FUNCTION_BLOCK PUBLIC FB_Observable IMPLEMENTS I_Observable
VAR_INPUT
	iParent:		I_Element;	
END_VAR
VAR
	bObserver:		BOOL;
	pList: 			POINTER TO I_Element;
    {attribute 'hide'}
	nLength:		DINT;
	{IF (defined (release))}
    	{attribute 'hide'}
	{END_IF}
	aList:			POINTER TO POINTER TO ARRAY [0..100] OF I_Element:=ADR(pList);
END_VAR

// https://peterzerlauth.com/
bObserver:= TRUE;

METHOD FB_exit : BOOL
VAR_INPUT
	bInCopyCode : BOOL; // if TRUE, the exit method is called for exiting an instance that is copied afterwards (online change).
END_VAR
M_Clear();
END_METHOD

METHOD M_Attach : BOOL
VAR_INPUT
	iObject: 	I_Element;
END_VAR
VAR
	pOldList: 	POINTER TO I_Element;
END_VAR
IF iObject <> 0 THEN
	// First Item
	IF pList = 0 THEN
		nLength:= nLength + 1;
		pList:= __NEW(POINTER TO I_Element,DINT_TO_UDINT(nLength));
	ELSE
		// Item already in List
		IF M_Find(iObject) = -1 THEN
			// backup 
			pOldList:= pList;
			// new Length
			nLength:= nLength + 1;
			// new pointer
			pList:= __NEW(POINTER TO I_Element,DINT_TO_UDINT(nLength));
			// restore
			Memcpy(pList,pOldList, SIZEOF(POINTER TO I_Element)*DINT_TO_UDINT(nLength -1));
			// delete old
			__DELETE(pOldList);
		ELSE
			M_Attach:= FALSE;	
			RETURN;
		END_IF
	END_IF
	IF pList = 0 THEN
		RETURN;
	END_IF
	// add new Object
	pList[nLength-1]:= iObject;
	M_Attach:= TRUE;
ELSE
	M_Attach:= FALSE;	
END_IF
END_METHOD

METHOD M_Clear
IF pList <> 0 THEN
	nLength:= 0;
	__DELETE(pList);
END_IF
END_METHOD

METHOD M_Detach : BOOL
VAR_INPUT
	iObject: 	I_Element;
END_VAR
VAR
	pOldList:			POINTER TO I_Element;
	nPosition: 			DINT;
END_VAR
IF iObject <> 0 THEN
	// First Item
	IF nLength >= 0 THEN
		// Item already in List
		nPosition:= M_Find(iObject);
		IF nPosition <> -1 THEN
			// backup 
			pOldList:= pList;
			// new Length
			nLength:= nLength -1;
			// new pointer
			pList:= __NEW(POINTER TO I_Element,DINT_TO_UDINT(nLength));
			// restore lower part
			Memcpy(pList,pOldList, SIZEOF(POINTER TO I_Element) * DINT_TO_UDINT(nPosition));
			//pList[nPosition]:= iObject;
			Memcpy(pList + (SIZEOF(POINTER TO I_Element)*nPosition),pOldList + (SIZEOF(POINTER TO I_Element)*(nPosition + 1)), SIZEOF(POINTER TO I_Element) * DINT_TO_UDINT(nLength - nPosition));
			// delete old
			__DELETE(pOldList);
		ELSE
			M_Detach:= FALSE;	
			RETURN;
		END_IF
	ELSE
		M_Detach:= FALSE;	
		RETURN;
	END_IF
	M_Detach:= TRUE;
ELSE
	M_Detach:= FALSE;	
END_IF
END_METHOD

METHOD M_Find : DINT
VAR_INPUT
	iObject: 	I_Element;
END_VAR
VAR
	nIndex: 	UINT;
END_VAR
// Object already in List
M_Find := -1;
WHILE nIndex < nLength DO
    IF (pList[nIndex] = iObject) THEN
        M_Find := nIndex;
        RETURN;
    END_IF
	nIndex := nIndex + 1;
END_WHILE
END_METHOD

METHOD M_Index : I_Observer
VAR_INPUT
	nIndex: 	DINT;
END_VAR
IF nIndex <= nLength THEN
	M_Index:= pList[nIndex].P_Event.P_Observer;
END_IF
END_METHOD

METHOD M_Notify
VAR_INPUT
	iSender:		I_Element;
END_VAR

VAR
	nIndex: 		DINT;
END_VAR
iParent.M_Request(E_Request.Abort);
IF bObserver THEN
	bObserver:= FALSE;
	WHILE nIndex < nLength DO
		pList[nIndex].P_Event.P_Observer.M_Notify(iSender);	
		nIndex:= nIndex + 1; 
	END_WHILE
	
END_IF
END_METHOD

{attribute 'OPC.UA.DA.Property' := '1'}
{attribute 'monitoring' := 'call'}
PROPERTY P_Length : DINT
GET
P_Length:= nLength;
END_GET
END_PROPERTY

END_FUNCTION_BLOCK

(* stored: Version 1.1.0.1
   POU FB_Observable: Id {52aee6c6-b98c-4cb9-9b9b-2f523841c4cc}, SpecialFunc None
   Method FB_exit: Id {8920c8e0-5709-4e5e-a21f-0871704cdcd1}
   Method M_Attach: Id {a96df4cc-8cea-4396-beb7-115ce888674b}
   Method M_Clear: Id {307f5dd9-2a35-4b04-93bb-a7de0406e653}
   Method M_Detach: Id {6e982e5c-8b12-4999-bbf2-06e2eebe2934}
   Method M_Find: Id {315829c2-37f1-487f-acb0-fff200e1a3d8}
   Method M_Index: Id {6e332950-284b-4ced-bcaa-31bfc1d4668b}
   Method M_Notify: Id {3d3fb67b-dd6a-440b-9c1c-e8b43c7588bf}
   Property P_Length: Id {8da11863-b503-4855-a3f1-c1f64dac07a1}
   Get Get: Id {81573980-0484-490c-84fc-be91d0b14826} *)
